Universal Robots URScript: 00B_01_ZhuaXian.script

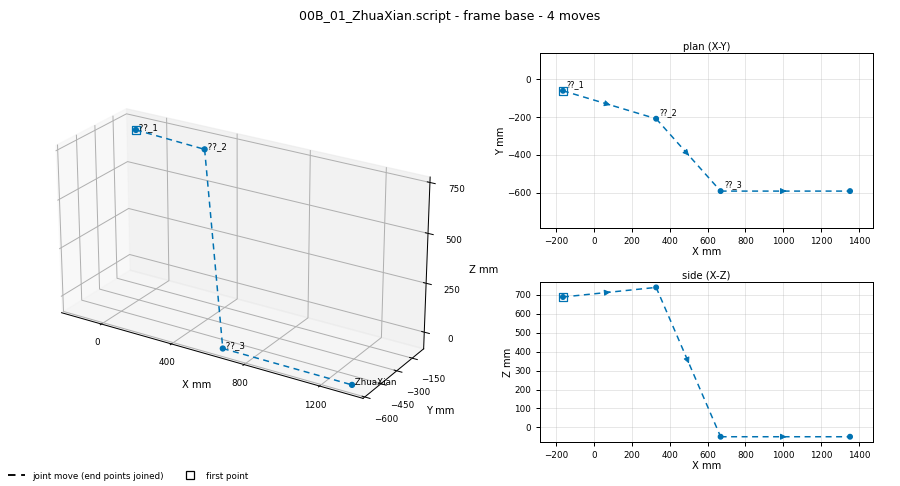
[picture p0: tool path of 00B_01_ZhuaXian.script in frame base, 4 of 4 moves have a stored position in this frame; points joined in program order, loops and branches not executed]
def P00B_01_ZhuaXian():
  set_gravity([0.0, 0.0, 9.82])
  set_safety_mode_transition_hardness(1)
  set_standard_analog_input_domain(0, 1)
  set_standard_analog_input_domain(1, 1)
  set_tool_analog_input_domain(0, 1)
  set_tool_analog_input_domain(1, 1)
  set_analog_outputdomain(0, 0)
  set_analog_outputdomain(1, 0)
  set_tool_voltage(24)
  set_input_actions_to_default()
  set_tcp(p[0.0,0.0,0.32,0.0,0.0,-0.5236])
  set_payload(0.0)
  global Zhua_1=[0.08063, -2.42649, -1.72682, -0.47876, 0.40808, -1.10831]
  global prepose=p[0.98979, -0.16931, -0.39963, 1.98720, 0.07234, 0.05469]
  global i_var_2=0
  global i_var_1=True
  global pose=p[0.98979, -0.31931, -0.39963, 1.98720, 0.07234, 0.05469]
  $ 1 "机器人程序"
  $ 2 "MoveJ"
  $ 3 "路点_1"
  set_tcp(p[0.0,0.0,0.32,0.0,0.0,-0.5236])
  movej(get_inverse_kin(p[-.163727558701, -.061396621977, .688653223316, .017033127778, .006361931554, -1.470657931683], qnear=[-1.5702031294452112, -2.7114549745732575E-4, -2.8754435221301478, -1.8534882704364222, -1.5660479704486292, -0.9517329374896448]), a=0.6981317007977318, v=0.5235987755982988)
  $ 4 "路点_2"
  set_tcp(p[0.0,0.0,0.32,0.0,0.0,-0.5236])
  movej(get_inverse_kin(p[.328392982749, -.208986586980, .739365657470, -.020049299877, .048647513572, -.078518253369], qnear=[-0.17769271532167608, -1.4830029646502894, -2.727104965840475, -0.5491274038897913, -1.6013763586627405, -0.9493606726275843]), a=0.6981317007977318, v=0.5235987755982988)
  $ 5 "路点_3"
  set_tcp(p[0.0,0.0,0.32,0.0,0.0,-0.5236])
  movej(get_inverse_kin(p[.668837031786, -.591204140121, -.049381654509, .134366608114, 1.558429351176, -.012521308084], qnear=[-0.9958465735064905, -2.235209290181295, -2.1793134848224085, -1.871134106312887, -2.477208439503805, -0.9766791502581995]), a=0.6981317007977318, v=0.5235987755982988)
  $ 6 "ZhuaXian"
  set_tcp(p[0.0,0.0,0.32,0.0,0.0,-0.5236])
  movej(get_inverse_kin(p[1.352436109272, -.591216839006, -.049372824621, .134324829362, 1.558483226668, -.012546260116], qnear=[-0.4123619238482874, -2.654867474232809, -1.1444781462298792, -2.4834540526019495, -1.8943169752704065, -0.9837244192706507]), a=0.6981317007977318, v=0.5235987755982988)
end
